# B&R Automation Studio project SoMRS_lab2
Automation Studio 4.5.2.102

## Configuration Config1

### Task classes (Cpu.sw)
```
Cyclic#2:
  Program <- Program.prg
Binaries: udbdef, TCData, ashwd, User, asfw, arconfig, sysconf, Role, ashwac, iomap
Libraries: MotorCtrl
```

## Logical view

### Program Logical/Program (ANSIC)

#### Init.c - Initialization code
```c
#include <bur/plctypes.h>

#ifdef _DEFAULT_INCLUDES
	#include <AsDefault.h>
#endif

void _INIT ProgramInit(void)
{
	fb_motor.dt=0.01; fb_motor.Ke=0.2; fb_motor.Tm=0.4; fb_motor.integrator.dt=0.01;
	fb_motor2.dt=0.01; fb_motor2.Ke=0.2; fb_motor2.Tm=0.4; fb_motor2.integrator.dt=0.01;

	fb_regulator.dt=0.01; fb_regulator.k_p=0.0064; fb_regulator.k_i=0.16; fb_regulator.max_abs_value=24; fb_regulator.integrator.dt=0.01;

	enable=1; count=0;
}
```

#### Cyclic.c
```c
#include <bur/plctypes.h>

#ifdef _DEFAULT_INCLUDES
	#include <AsDefault.h>
#endif

void _CYCLIC ProgramCyclic(void)
{
	if(enable)
	{
		count+=1; if(count<=50)
		{

		speed=50;
		}
		else
		{
			speed=0;

			 if(count>=100)
			{
				count=0;
			}
		}
	}
	fb_regulator.e=speed - fb_motor.w; fb_motor2.u=speed; FB_Regulator(&fb_regulator); fb_motor.u=fb_regulator.u; FB_Motor(&fb_motor); FB_Motor(&fb_motor2);
}
```

#### Variables.var - Local variables
```iecst
VAR
	speed : REAL;
	enable : BOOL;
	count : UINT;
	fb_motor2 : FB_Motor;
	fb_motor : FB_Motor;
	fb_regulator : FB_Regulator;
END_VAR
```

### Library Logical/MotorCtrl (ANSIC)

#### MotorCtrl.fun - Exported functions and function blocks
```iecst
FUNCTION_BLOCK FB_Integrator
	VAR_INPUT
		in : REAL; (*Вход*)
	END_VAR
	VAR_OUTPUT
		out : REAL; (*Выход*)
	END_VAR
	VAR
		dt : REAL; (*Частота дискретизации*)
		state : REAL; (*Предыдущее состояние двигателя*)
	END_VAR
END_FUNCTION_BLOCK

FUNCTION_BLOCK FB_Motor
	VAR_INPUT
		u : REAL; (*Вход Напряжение*)
	END_VAR
	VAR_OUTPUT
		w : REAL; (*Выход Обороты*)
	END_VAR
	VAR
		phi : REAL;
		integrator : FB_Integrator; (*ФБ интегратора*)
		Tm : REAL;
		Ke : REAL;
		dt : REAL;
	END_VAR
END_FUNCTION_BLOCK

FUNCTION_BLOCK FB_Regulator
	VAR_INPUT
		e : REAL;
	END_VAR
	VAR_OUTPUT
		u : REAL;
	END_VAR
	VAR
		k_p : REAL;
		k_i : REAL;
		integrator : FB_Integrator;
		iyOld : REAL;
		max_abs_value : REAL;
		dt : REAL;
		e_kp : REAL;
	END_VAR
END_FUNCTION_BLOCK
```

#### FB_Integrator.c - Cyclic code
```c
#include <bur/plctypes.h>

#ifdef _DEFAULT_INCLUDES
	#include <AsDefault.h>
#endif

void FB_Integrator(struct FB_Integrator* inst)
{
	inst->out = inst->dt * inst ->in + inst ->state;
	inst ->state = inst ->out;
}
```

#### FB_Motor.c
```c
#include <bur/plctypes.h>

#ifdef _DEFAULT_INCLUDES
	#include <AsDefault.h>
#endif

void FB_Motor(struct FB_Motor* inst)
{
	REAL a = inst->u / inst->Ke - inst->phi;
	REAL w = a / inst ->Tm;
	inst ->integrator.in = w;
	FB_Integrator(&inst->integrator);
	inst ->phi = inst->integrator.out;

/*	inst->integrator.in=(inst->u/inst->Ke-inst->w)*inst->dt/inst->Tm;
	inst->integrator.out=inst->w;
	FB_Integrator(&(inst->integrator));
	inst->w=inst->integrator.out;
	inst->integrator.in=inst->w*inst->dt;
	inst->integrator.out=inst->phi;
	FB_Integrator(&(inst->integrator));
	inst->phi=inst->integrator.out;*/
}
```

#### FB_Regulator.c
```c
#include <bur/plctypes.h>

#ifdef _DEFAULT_INCLUDES
	#include <AsDefault.h>
#endif

void FB_Regulator(struct FB_Regulator* inst)
{
	inst->integrator.in=inst->e * inst->k_i * inst->dt + inst->iyOld; FB_Integrator(&(inst->integrator)); inst->e_kp=inst->e*inst->k_p;
	inst->e_kp=(inst->e_kp > inst->max_abs_value || inst->e_kp < - inst->max_abs_value)?((inst->e_kp>0)?inst->max_abs_value:-inst->max_abs_value):inst->e_kp; inst->e_kp+=inst->integrator.out;
	inst->u=(inst->e_kp > inst->max_abs_value || inst->e_kp < - inst->max_abs_value)?((inst->e_kp>0)?inst->max_abs_value:-inst->max_abs_value):inst->e_kp; inst->iyOld=inst->u-inst->e_kp;
}
```

Listed in the project but not available here: Logical/Global.typ, Logical/Global.var, Logical/Libraries, Logical/Program/Exit.c, Logical/Program/Types.typ, Logical/MotorCtrl/Types.typ, Logical/MotorCtrl/Constants.var
